(* IEC 61131-3 sources: test/Class/Sfc_Logic_Or_3, 1 file *)

(* ---- Sfc_Logic_Or_3.st ---- *)
(*!
<Class
	Name               = "Sfc_Logic_Or_3"
	Revision           = "1.1"
	RealtimeTask       = "false"
	CyclicTask         = "false"
	BackgroundTask     = "false"
	Sigmatek           = "true"
	OSInterface        = "false"
	HighPriority       = "false"
	Automatic          = "false"
	UpdateMode         = "Prescan"
	IconPath           = ".\Class\Sfc_Logic_Or_3\Logic_Or_Base.ico"
	SharedCommandTable = "true"
	Objectsize         = "(284,120)"
	Comment            = "V1.1 Logic OR class with 3 operands">
	<Channels>
		<Server
			Name           = "Result"
			Initialize     = "false"
			Visualized     = "false"
			WriteProtected = "true"
			Comment        = "If one client is &lt;&gt; 0 then result = 1">
		</Server>
		<Client Name="Op1" Required="false" Internal="false" Comment="Operand 1"/>
		<Client Name="Op2" Required="false" Internal="false" Comment="Operand 2"/>
		<Client Name="Op3" Required="false" Internal="false" Comment="Operand 3"/>
	</Channels>
	<Network Name="Sfc_Logic_Or_3">
		<!-- List of Components in this network -->
		<Components>
			<Object
				Name       = "_base"
				Class      = "Sfc_Logic_Or_Base"
				Position   = "(420,750)"
				Visualized = "false">
				<Channels>
					<Server Name="Result"/>
				</Channels>
			</Object>
		</Components>
		<Comments>
		</Comments>
		<!-- List of Connections in this network -->
		<Connections>
			<Connection Source="this.Result" Destination="_base.Result" Vertices="(892,210),(720,840),"/>
		</Connections>
		<!-- Headerfiles -->
		<Options>
		</Options>
	</Network>
</Class>
*)
#pragma using Sfc_Logic_Or_Base

Sfc_Logic_Or_3 : CLASS
: Sfc_Logic_Or_Base
  //Servers:
  //Clients:
	Op1 	: CltCh_DINT;
	Op2 	: CltCh_DINT;
	Op3 	: CltCh_DINT;
  //Variables:
  //Functions:
  //Tables:
	FUNCTION @STD
		VAR_OUTPUT
			ret_code	: CONFSTATES;
		END_VAR;
	FUNCTION GLOBAL TAB @CT_;
END_CLASS;
